INTERFACE I_Execution

METHOD Abort 
VAR_INPUT
END_VAR
END_METHOD

PROPERTY Aborted : BOOL
GET
END_GET
END_PROPERTY

PROPERTY Busy : BOOL
GET
END_GET
END_PROPERTY

METHOD Clear 
VAR_INPUT
END_VAR
END_METHOD

PROPERTY Done : BOOL
GET
END_GET
END_PROPERTY

PROPERTY Error : BOOL
GET
END_GET
END_PROPERTY

PROPERTY ErrorMsg : T_MaxString
GET
END_GET
SET
END_SET
END_PROPERTY

PROPERTY Notification_OnAbort : I_Notification
GET
END_GET
SET
END_SET
END_PROPERTY

PROPERTY Notification_OnError : I_Notification
GET
END_GET
SET
END_SET
END_PROPERTY

PROPERTY Ready : BOOL
GET
END_GET
END_PROPERTY

METHOD Start : BOOL // returns TRUE if start request accepted (i.e State was Ready)
VAR_INPUT
END_VAR
END_METHOD

PROPERTY Starting : BOOL
GET
END_GET
END_PROPERTY

END_INTERFACE

(* stored: Version 1.1.0.1, ProductVersion 3.1.4024.6
   Itf I_Execution: Id {2e2a9e90-2894-0caa-065e-86441183945f}
   Folder Methods: Id {4df2c49f-ecc5-41ac-a5f7-eb029ec847e7}
   Folder Properties: Id {858ea4b7-fbd7-4d4c-a650-4ab711825959}
   Method Abort: Id {b913466c-26cf-0433-3b1e-51d91dedf168}
   Property Aborted: Id {5347566a-e4a6-4028-bbdd-c7c385fe1cab}
   Get Get: Id {68b612a5-196e-4381-a504-106ddf11c80e}
   Property Busy: Id {6cebbaf7-86c1-4b42-b741-1563ee9a82a3}
   Get Get: Id {c2417d08-69f5-4b45-8674-471ac6e75ca8}
   Method Clear: Id {58de2a78-426c-4017-a46d-fddd798e420e}
   Property Done: Id {f19ffc53-eaf1-48be-aca7-f281232899dc}
   Get Get: Id {06415348-1825-402b-9b90-995ba15a6503}
   Property Error: Id {54cfaecc-395a-4685-8d6b-701b343961c9}
   Get Get: Id {cff8eb45-644a-457e-91bd-f88883679daa}
   Property ErrorMsg: Id {1d2434d1-a947-47bc-b679-2969b90c75f0}
   Get Get: Id {fc1803ed-3692-454e-89f2-239f5db0e4f9}
   Set Set: Id {0f8e317d-22aa-45ae-9919-ecca1a28a96e}
   Property Notification_OnAbort: Id {5bff5e48-e058-4bd5-b034-78e58ed48528}
   Get Get: Id {2d849f1f-c182-4380-910a-ae92c4aa8e38}
   Set Set: Id {f7c5526a-9c46-4575-b20a-013d7f3bf3a6}
   Property Notification_OnError: Id {b1fef8e3-b1dc-4f81-ad00-3f9ccb825c81}
   Get Get: Id {e6794e2f-7391-458f-a3be-a68c40a6b2fb}
   Set Set: Id {8f58c853-4be2-45e4-a65e-1a6be90df3b5}
   Property Ready: Id {b91ada47-a851-4255-ace3-07ff2a4d3deb}
   Get Get: Id {bde8a44c-e6cd-483a-a94e-c0d4f73a98b1}
   Method Start: Id {28e25cff-ad88-0708-05e8-5a4e484e10dc}
   Property Starting: Id {6b02f8f3-9828-4ea0-8253-65483424421e}
   Get Get: Id {d6faa71d-a2a3-4abf-8c36-46cccd4f90e4} *)
